// TIA Portal project "AUTOMATED_AIR_CONDITION" (V15)

(* hardware
DEVICE "S7-1200 station_1"  S7-1200 Station
   slot 0: "Rack_0"  S7-1200 Rack  Rack  V1.0
   slot 1: "PLC_1"  CPU 1214C DC/DC/DC  6ES7 214-1AG40-0XB0  V4.2
*)

// ===== PLC "PLC_1"  CPU 1214C DC/DC/DC =====

VAR_GLOBAL   // PLC tag table "Default tag table"
   "Clock_Byte" AT %MB80 : Byte;
   "Clock_10Hz" AT %M80.0 : Bool;
   "Clock_5Hz" AT %M80.1 : Bool;
   "Clock_2.5Hz" AT %M80.2 : Bool;
   "Clock_2Hz" AT %M80.3 : Bool;
   "Clock_1.25Hz" AT %M80.4 : Bool;
   "Clock_1Hz" AT %M80.5 : Bool;
   "Clock_0.625Hz" AT %M80.6 : Bool;
   "Clock_0.5Hz" AT %M80.7 : Bool;
   "Tag_18" AT %M20.0 : Bool;
   "Tag_19" AT %M20.1 : Bool;
   "Tag_3" AT %Q0.0 : Bool;
   "Tag_5" AT %MD12 : Real;
   "Error" AT %MW70 : Int;
   "temp" AT %MD10 : Real;
END_VAR

ORGANIZATION_BLOCK "Main"   // OB1, LAD, ProgramCycle
TITLE = "Main Program Sweep (Cycle)"
{ S7_Optimized_Access := 'TRUE' }
VERSION : 0.1
   VAR_INPUT
      Initial_Call : Bool;   // Initial call of this OB
      Remanence : Bool;   // =True, if remanent data are available
   END_VAR
BEGIN

REGION Network 1
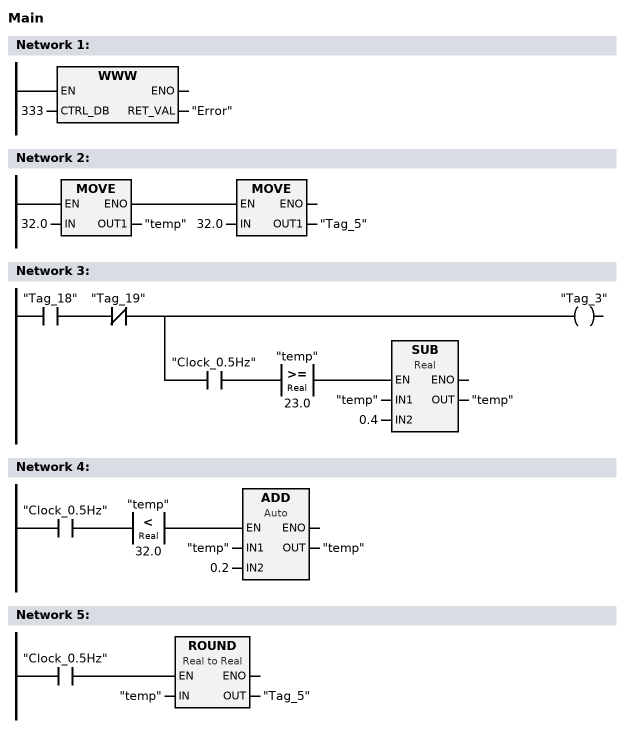
   "Error" := WWW(CTRL_DB := 333);
END_REGION

REGION Network 2
   RUNG wire#powerrail
      Move(in := 32.0, out1 => "temp")
      Move(in := 32.0, out1 => "Tag_5")
   END_RUNG
   // the same network as SCL:
   "temp" := 32.0;
   "Tag_5" := 32.0;
END_REGION

REGION Network 3
   RUNG wire#powerrail
      Contact( "Tag_18" )
      I_Contact( "Tag_19" )
      wire#w1
      Coil( "Tag_3" )
   END_RUNG
   RUNG wire#w1
      Contact( "Clock_0.5Hz" )
      { S7_Templates := "SrcType := Real" } GE_Contact(in1 := "temp", in2 := 23.0)
      { S7_Templates := "SrcType := Real" } Sub(in1 := "temp", in2 := 0.4, out => "temp")
   END_RUNG
   // the same network as SCL:
   "Tag_3" := "Tag_18" AND NOT "Tag_19";
   IF "Tag_3" AND "Clock_0.5Hz" AND ("temp" >= 23.0) THEN "temp" := "temp" - 0.4; END_IF;
END_REGION

REGION Network 4
   RUNG wire#powerrail
      Contact( "Clock_0.5Hz" )
      { S7_Templates := "SrcType := Real" } LT_Contact(in1 := "temp", in2 := 32.0)
      Add(in1 := "temp", in2 := 0.2, out => "temp")
   END_RUNG
   // the same network as SCL:
   IF "Clock_0.5Hz" AND ("temp" < 32.0) THEN "temp" := "temp" + 0.2; END_IF;
END_REGION

REGION Network 5
   RUNG wire#powerrail
      Contact( "Clock_0.5Hz" )
      { S7_Templates := "[SrcType := Real, DestType := Real]" } Round(in := "temp", out => "Tag_5")
   END_RUNG
   // the same network as SCL:
   IF "Clock_0.5Hz" THEN "Tag_5" := ROUND("temp"); END_IF;
END_REGION
END_ORGANIZATION_BLOCK